PROGRAM MAIN_1
VAR
	fbEventlogger : FB_TcEventLogger;
	fbAlarm: FB_TcAlarm;
	fbMessage: FB_TcMessage;
	
	bAlarm: BOOL;
	bMessage : BOOL;
	bIsInitalized: BOOL;
	bClearAlarm: BOOL;
	bConfirmAlarm: BOOL;
END_VAR

IF NOT bIsInitalized THEN
	bIsInitalized := TRUE;
	fbMessage.CreateEx(TC_Events.MyEvents.Start, 0);
	fbAlarm.CreateEx(TC_Events.MyEvents.Stop, TRUE, 0);
END_IF

IF bMessage THEN
	bMessage := FALSE;
	fbMessage.Send(0);
END_IF

IF bAlarm THEN
	bAlarm := FALSE;
	fbAlarm.Raise(0);
END_IF

IF bClearAlarm THEN
	bClearAlarm := FALSE;
	fbAlarm.Clear(0, TRUE);
END_IF

END_PROGRAM

(* stored: Version 1.1.0.1, ProductVersion 3.1.4024.4
   POU MAIN_1: Id {9ae84a09-de24-4b52-a2ed-2baa5985f4b1}, SpecialFunc None *)
